// TIA Portal V15.1 export
// export: Created 2024-06-21T08:41:02.9041291Z, ExportSetting WithDefaults, DisplayName Totally Integrated Automation Portal, DisplayVersion V15.1 Update 5, DisplayName TIA Portal Openness, DisplayVersion V15.1 Update 5, DisplayName SINAMICS Startdrive Advanced, DisplayVersion V15.1, DisplayName G130, G150, S120, S150, SINAMICS MV, S210, DisplayVersion V15.1, DisplayName G110M, G120, G120C, G120D, G120P, DisplayVersion V15.1, DisplayName STEP 7 Professional, DisplayVersion V15.1 Update 5, DisplayName STEP 7 Safety, DisplayVersion V15.1, DisplayName WinCC Professional, DisplayVersion V15.1 Update 5, DisplayName SIMATIC Visualization Architect, DisplayVersion V15.1
FUNCTION_BLOCK "LProcModesSum"   // FB1702, FBD
TITLE = LProcModesSum
{ S7_Optimized_Access := 'FALSE' }
AUTHOR : VCC
FAMILY : ProcEqp
NAME : ModesSum
VERSION : 1.0
// ================================================================================
// Create the Modes Summary for 20 possible components
// ================================================================================
// stored: AutoNumber false, IsIECCheckEnabled false, SetENOAutomatically False, UDAEnableTagReadback false
   VAR_INPUT
      I_StartPB { ExternalAccessible := 'False'; ExternalVisible := 'False'; ExternalWritable := 'False'} : Bool;   // Summary of Start buttons
      I_AlarmResetPB { ExternalAccessible := 'False'; ExternalVisible := 'False'; ExternalWritable := 'False'} : Bool;   // Summary of Alarm reset buttons
      I_SafetyNotOk { ExternalAccessible := 'False'; ExternalVisible := 'False'; ExternalWritable := 'False'} : Bool;   // Safety is not ok
      I_ObjectMode1 { ExternalAccessible := 'False'; ExternalVisible := 'False'; ExternalWritable := 'False'} : Word;   // Modes Component 1
      I_ObjectMode2 { ExternalAccessible := 'False'; ExternalVisible := 'False'; ExternalWritable := 'False'} : Word;   // Modes Component 2
      I_ObjectMode3 { ExternalAccessible := 'False'; ExternalVisible := 'False'; ExternalWritable := 'False'} : Word;   // Modes Component 3
      I_ObjectMode3Used { ExternalAccessible := 'False'; ExternalVisible := 'False'; ExternalWritable := 'False'} : Bool;   // True if used
      I_ObjectMode4 { ExternalAccessible := 'False'; ExternalVisible := 'False'; ExternalWritable := 'False'} : Word;   // Modes Component 4
      I_ObjectMode4Used { ExternalAccessible := 'False'; ExternalVisible := 'False'; ExternalWritable := 'False'} : Bool;   // True if used
      I_ObjectMode5 { ExternalAccessible := 'False'; ExternalVisible := 'False'; ExternalWritable := 'False'} : Word;   // Modes Component 5
      I_ObjectMode5Used { ExternalAccessible := 'False'; ExternalVisible := 'False'; ExternalWritable := 'False'} : Bool;   // True if used
      I_ObjectMode6 { ExternalAccessible := 'False'; ExternalVisible := 'False'; ExternalWritable := 'False'} : Word;   // Modes Component 6
      I_ObjectMode6Used { ExternalAccessible := 'False'; ExternalVisible := 'False'; ExternalWritable := 'False'} : Bool;   // True if used
      I_ObjectMode7 { ExternalAccessible := 'False'; ExternalVisible := 'False'; ExternalWritable := 'False'} : Word;   // Modes Component 7
      I_ObjectMode7Used { ExternalAccessible := 'False'; ExternalVisible := 'False'; ExternalWritable := 'False'} : Bool;   // True if used
      I_ObjectMode8 { ExternalAccessible := 'False'; ExternalVisible := 'False'; ExternalWritable := 'False'} : Word;   // Modes Component 8
      I_ObjectMode8Used { ExternalAccessible := 'False'; ExternalVisible := 'False'; ExternalWritable := 'False'} : Bool;   // True if used
      I_ObjectMode9 { ExternalAccessible := 'False'; ExternalVisible := 'False'; ExternalWritable := 'False'} : Word;   // Modes Component 9
      I_ObjectMode9Used { ExternalAccessible := 'False'; ExternalVisible := 'False'; ExternalWritable := 'False'} : Bool;   // True if used
      I_ObjectMode10 { ExternalAccessible := 'False'; ExternalVisible := 'False'; ExternalWritable := 'False'} : Word;   // Modes Component 10
      I_ObjectMode10Used { ExternalAccessible := 'False'; ExternalVisible := 'False'; ExternalWritable := 'False'} : Bool;   // True if used
      I_ObjectMode11 { ExternalAccessible := 'False'; ExternalVisible := 'False'; ExternalWritable := 'False'} : Word;   // Modes Component 11
      I_ObjectMode11Used { ExternalAccessible := 'False'; ExternalVisible := 'False'; ExternalWritable := 'False'} : Bool;   // True if used
      I_ObjectMode12 { ExternalAccessible := 'False'; ExternalVisible := 'False'; ExternalWritable := 'False'} : Word;   // Modes Component 12
      I_ObjectMode12Used { ExternalAccessible := 'False'; ExternalVisible := 'False'; ExternalWritable := 'False'} : Bool;   // True if used
      I_ObjectMode13 { ExternalAccessible := 'False'; ExternalVisible := 'False'; ExternalWritable := 'False'} : Word;   // Modes Component 13
      I_ObjectMode13Used { ExternalAccessible := 'False'; ExternalVisible := 'False'; ExternalWritable := 'False'} : Bool;   // True if used
      I_ObjectMode14 { ExternalAccessible := 'False'; ExternalVisible := 'False'; ExternalWritable := 'False'} : Word;   // Modes Component 14
      I_ObjectMode14Used { ExternalAccessible := 'False'; ExternalVisible := 'False'; ExternalWritable := 'False'} : Bool;   // True if used
      I_ObjectMode15 { ExternalAccessible := 'False'; ExternalVisible := 'False'; ExternalWritable := 'False'} : Word;   // Modes Component 15
      I_ObjectMode15Used { ExternalAccessible := 'False'; ExternalVisible := 'False'; ExternalWritable := 'False'} : Bool;   // True if used
      I_ObjectMode16 { ExternalAccessible := 'False'; ExternalVisible := 'False'; ExternalWritable := 'False'} : Word;   // Modes Component 16
      I_ObjectMode16Used { ExternalAccessible := 'False'; ExternalVisible := 'False'; ExternalWritable := 'False'} : Bool;   // True if used
      I_ObjectMode17 { ExternalAccessible := 'False'; ExternalVisible := 'False'; ExternalWritable := 'False'} : Word;   // Modes Component 17
      I_ObjectMode17Used { ExternalAccessible := 'False'; ExternalVisible := 'False'; ExternalWritable := 'False'} : Bool;   // True if used
      I_ObjectMode18 { ExternalAccessible := 'False'; ExternalVisible := 'False'; ExternalWritable := 'False'} : Word;   // Modes Component 18
      I_ObjectMode18Used { ExternalAccessible := 'False'; ExternalVisible := 'False'; ExternalWritable := 'False'} : Bool;   // True if used
      I_ObjectMode19 { ExternalAccessible := 'False'; ExternalVisible := 'False'; ExternalWritable := 'False'} : Word;   // Modes Component 19
      I_ObjectMode19Used { ExternalAccessible := 'False'; ExternalVisible := 'False'; ExternalWritable := 'False'} : Bool;   // True if used
      I_ObjectMode20 { ExternalAccessible := 'False'; ExternalVisible := 'False'; ExternalWritable := 'False'} : Word;   // Modes Component 20
      I_ObjectMode20Used { ExternalAccessible := 'False'; ExternalVisible := 'False'; ExternalWritable := 'False'} : Bool;   // True if used
   END_VAR
   VAR_OUTPUT
      O_AutoSel { ExternalAccessible := 'False'; ExternalVisible := 'False'; ExternalWritable := 'False'} : Bool;   // At least one component is in auto selected
      O_Auto { ExternalAccessible := 'False'; ExternalVisible := 'False'; ExternalWritable := 'False'} : Bool;   // All the components are in auto
      O_ManSel { ExternalAccessible := 'False'; ExternalVisible := 'False'; ExternalWritable := 'False'} : Bool;   // At least one component is in manual selected
      O_Man { ExternalAccessible := 'False'; ExternalVisible := 'False'; ExternalWritable := 'False'} : Bool;   // At least one component is in manual
      O_AlarmResetPB { ExternalAccessible := 'False'; ExternalVisible := 'False'; ExternalWritable := 'False'} : Bool;   // Alarm reset button is activated
   END_VAR
   VAR DB_SPECIFIC
      H_Anim : Word;   // Mode Animation Word
      H_Anim2 : Word;   // Mode Animation Word
      H_ConfigBtnResetTM : Bool;   // From the HMI - Config internal tag
      H_ConfigBtnResetSeq : Bool;   // From the HMI - Config internal tag
      H_ModeChanged : Bool;   // From the HMI - Mode changed to Auto
      H_ScreenChanged : Bool;   // From the HMI - The screen has changed
      AutoSel1 { ExternalAccessible := 'False'; ExternalVisible := 'False'; ExternalWritable := 'False'} : Bool;   // Auto selected Component 1
      Auto1 { ExternalAccessible := 'False'; ExternalVisible := 'False'; ExternalWritable := 'False'} : Bool;   // Auto Component 1
      ManSel1 { ExternalAccessible := 'False'; ExternalVisible := 'False'; ExternalWritable := 'False'} : Bool;   // Manu selected Component 1
      Man1 { ExternalAccessible := 'False'; ExternalVisible := 'False'; ExternalWritable := 'False'} : Bool;   // Manu Component 1
      AutoSel2 { ExternalAccessible := 'False'; ExternalVisible := 'False'; ExternalWritable := 'False'} : Bool;   // Auto selected Component 2
      Auto2 { ExternalAccessible := 'False'; ExternalVisible := 'False'; ExternalWritable := 'False'} : Bool;   // Auto Component 2
      ManSel2 { ExternalAccessible := 'False'; ExternalVisible := 'False'; ExternalWritable := 'False'} : Bool;   // Manu selected Component 2
      Man2 { ExternalAccessible := 'False'; ExternalVisible := 'False'; ExternalWritable := 'False'} : Bool;   // Manu Component 2
      AutoSel3 { ExternalAccessible := 'False'; ExternalVisible := 'False'; ExternalWritable := 'False'} : Bool;   // Auto selected Component 3
      Auto3 { ExternalAccessible := 'False'; ExternalVisible := 'False'; ExternalWritable := 'False'} : Bool;   // Auto Component 3
      ManSel3 { ExternalAccessible := 'False'; ExternalVisible := 'False'; ExternalWritable := 'False'} : Bool;   // Manu selected Component 3
      Man3 { ExternalAccessible := 'False'; ExternalVisible := 'False'; ExternalWritable := 'False'} : Bool;   // Manu Component 3
      AutoSel4 { ExternalAccessible := 'False'; ExternalVisible := 'False'; ExternalWritable := 'False'} : Bool;   // Auto selected Component 4
      Auto4 { ExternalAccessible := 'False'; ExternalVisible := 'False'; ExternalWritable := 'False'} : Bool;   // Auto Component 4
      ManSel4 { ExternalAccessible := 'False'; ExternalVisible := 'False'; ExternalWritable := 'False'} : Bool;   // Manu selected Component 4
      Man4 { ExternalAccessible := 'False'; ExternalVisible := 'False'; ExternalWritable := 'False'} : Bool;   // Manu Component 4
      AutoSel5 { ExternalAccessible := 'False'; ExternalVisible := 'False'; ExternalWritable := 'False'} : Bool;   // Auto selected Component 5
      Auto5 { ExternalAccessible := 'False'; ExternalVisible := 'False'; ExternalWritable := 'False'} : Bool;   // Auto Component 5
      ManSel5 { ExternalAccessible := 'False'; ExternalVisible := 'False'; ExternalWritable := 'False'} : Bool;   // Manu selected Component 5
      Man5 { ExternalAccessible := 'False'; ExternalVisible := 'False'; ExternalWritable := 'False'} : Bool;   // Manu Component 5
      AutoSel6 { ExternalAccessible := 'False'; ExternalVisible := 'False'; ExternalWritable := 'False'} : Bool;   // Auto selected Component 6
      Auto6 { ExternalAccessible := 'False'; ExternalVisible := 'False'; ExternalWritable := 'False'} : Bool;   // Auto Component 6
      ManSel6 { ExternalAccessible := 'False'; ExternalVisible := 'False'; ExternalWritable := 'False'} : Bool;   // Manu selected Component 6
      Man6 { ExternalAccessible := 'False'; ExternalVisible := 'False'; ExternalWritable := 'False'} : Bool;   // Manu Component 6
      AutoSel7 { ExternalAccessible := 'False'; ExternalVisible := 'False'; ExternalWritable := 'False'} : Bool;   // Auto selected Component 7
      Auto7 { ExternalAccessible := 'False'; ExternalVisible := 'False'; ExternalWritable := 'False'} : Bool;   // Auto Component 7
      ManSel7 { ExternalAccessible := 'False'; ExternalVisible := 'False'; ExternalWritable := 'False'} : Bool;   // Manu selected Component 7
      Man7 { ExternalAccessible := 'False'; ExternalVisible := 'False'; ExternalWritable := 'False'} : Bool;   // Manu Component 7
      AutoSel8 { ExternalAccessible := 'False'; ExternalVisible := 'False'; ExternalWritable := 'False'} : Bool;   // Auto selected Component 8
      Auto8 { ExternalAccessible := 'False'; ExternalVisible := 'False'; ExternalWritable := 'False'} : Bool;   // Auto Component 8
      ManSel8 { ExternalAccessible := 'False'; ExternalVisible := 'False'; ExternalWritable := 'False'} : Bool;   // Manu selected Component 8
      Man8 { ExternalAccessible := 'False'; ExternalVisible := 'False'; ExternalWritable := 'False'} : Bool;   // Manu Component 8
      AutoSel9 { ExternalAccessible := 'False'; ExternalVisible := 'False'; ExternalWritable := 'False'} : Bool;   // Auto selected Component 9
      Auto9 { ExternalAccessible := 'False'; ExternalVisible := 'False'; ExternalWritable := 'False'} : Bool;   // Auto Component 9
      ManSel9 { ExternalAccessible := 'False'; ExternalVisible := 'False'; ExternalWritable := 'False'} : Bool;   // Manu selected Component 9
      Man9 { ExternalAccessible := 'False'; ExternalVisible := 'False'; ExternalWritable := 'False'} : Bool;   // Manu Component 9
      AutoSel10 { ExternalAccessible := 'False'; ExternalVisible := 'False'; ExternalWritable := 'False'} : Bool;   // Auto selected Component 10
      Auto10 { ExternalAccessible := 'False'; ExternalVisible := 'False'; ExternalWritable := 'False'} : Bool;   // Auto Component 10
      ManSel10 { ExternalAccessible := 'False'; ExternalVisible := 'False'; ExternalWritable := 'False'} : Bool;   // Manu selected Component 10
      Man10 { ExternalAccessible := 'False'; ExternalVisible := 'False'; ExternalWritable := 'False'} : Bool;   // Manu Component 10
      AutoSel11 { ExternalAccessible := 'False'; ExternalVisible := 'False'; ExternalWritable := 'False'} : Bool;   // Auto selected Component 11
      Auto11 { ExternalAccessible := 'False'; ExternalVisible := 'False'; ExternalWritable := 'False'} : Bool;   // Auto Component 11
      ManSel11 { ExternalAccessible := 'False'; ExternalVisible := 'False'; ExternalWritable := 'False'} : Bool;   // Manu selected Component 11
      Man11 { ExternalAccessible := 'False'; ExternalVisible := 'False'; ExternalWritable := 'False'} : Bool;   // Manu Component 11
      AutoSel12 { ExternalAccessible := 'False'; ExternalVisible := 'False'; ExternalWritable := 'False'} : Bool;   // Auto selected Component 12
      Auto12 { ExternalAccessible := 'False'; ExternalVisible := 'False'; ExternalWritable := 'False'} : Bool;   // Auto Component 12
      ManSel12 { ExternalAccessible := 'False'; ExternalVisible := 'False'; ExternalWritable := 'False'} : Bool;   // Manu selected Component 12
      Man12 { ExternalAccessible := 'False'; ExternalVisible := 'False'; ExternalWritable := 'False'} : Bool;   // Manu Component 12
      AutoSel13 { ExternalAccessible := 'False'; ExternalVisible := 'False'; ExternalWritable := 'False'} : Bool;   // Auto selected Component 13
      Auto13 { ExternalAccessible := 'False'; ExternalVisible := 'False'; ExternalWritable := 'False'} : Bool;   // Auto Component 13
      ManSel13 { ExternalAccessible := 'False'; ExternalVisible := 'False'; ExternalWritable := 'False'} : Bool;   // Manu selected Component 13
      Man13 { ExternalAccessible := 'False'; ExternalVisible := 'False'; ExternalWritable := 'False'} : Bool;   // Manu Component 13
      AutoSel14 { ExternalAccessible := 'False'; ExternalVisible := 'False'; ExternalWritable := 'False'} : Bool;   // Auto selected Component 14
      Auto14 { ExternalAccessible := 'False'; ExternalVisible := 'False'; ExternalWritable := 'False'} : Bool;   // Auto Component 14
      ManSel14 { ExternalAccessible := 'False'; ExternalVisible := 'False'; ExternalWritable := 'False'} : Bool;   // Manu selected Component 14
      Man14 { ExternalAccessible := 'False'; ExternalVisible := 'False'; ExternalWritable := 'False'} : Bool;   // Manu Component 14
      AutoSel15 { ExternalAccessible := 'False'; ExternalVisible := 'False'; ExternalWritable := 'False'} : Bool;   // Auto selected Component 15
      Auto15 { ExternalAccessible := 'False'; ExternalVisible := 'False'; ExternalWritable := 'False'} : Bool;   // Auto Component 15
      ManSel15 { ExternalAccessible := 'False'; ExternalVisible := 'False'; ExternalWritable := 'False'} : Bool;   // Manu selected Component 15
      Man15 { ExternalAccessible := 'False'; ExternalVisible := 'False'; ExternalWritable := 'False'} : Bool;   // Manu Component 15
      AutoSel16 { ExternalAccessible := 'False'; ExternalVisible := 'False'; ExternalWritable := 'False'} : Bool;   // Auto selected Component 16
      Auto16 { ExternalAccessible := 'False'; ExternalVisible := 'False'; ExternalWritable := 'False'} : Bool;   // Auto Component 16
      ManSel16 { ExternalAccessible := 'False'; ExternalVisible := 'False'; ExternalWritable := 'False'} : Bool;   // Manu selected Component 16
      Man16 { ExternalAccessible := 'False'; ExternalVisible := 'False'; ExternalWritable := 'False'} : Bool;   // Manu Component 16
      AutoSel17 { ExternalAccessible := 'False'; ExternalVisible := 'False'; ExternalWritable := 'False'} : Bool;   // Auto selected Component 17
      Auto17 { ExternalAccessible := 'False'; ExternalVisible := 'False'; ExternalWritable := 'False'} : Bool;   // Auto Component 17
      ManSel17 { ExternalAccessible := 'False'; ExternalVisible := 'False'; ExternalWritable := 'False'} : Bool;   // Manu selected Component 17
      Man17 { ExternalAccessible := 'False'; ExternalVisible := 'False'; ExternalWritable := 'False'} : Bool;   // Manu Component 17
      AutoSel18 { ExternalAccessible := 'False'; ExternalVisible := 'False'; ExternalWritable := 'False'} : Bool;   // Auto selected Component 18
      Auto18 { ExternalAccessible := 'False'; ExternalVisible := 'False'; ExternalWritable := 'False'} : Bool;   // Auto Component 18
      ManSel18 { ExternalAccessible := 'False'; ExternalVisible := 'False'; ExternalWritable := 'False'} : Bool;   // Manu selected Component 18
      Man18 { ExternalAccessible := 'False'; ExternalVisible := 'False'; ExternalWritable := 'False'} : Bool;   // Manu Component 18
      AutoSel19 { ExternalAccessible := 'False'; ExternalVisible := 'False'; ExternalWritable := 'False'} : Bool;   // Auto selected Component 19
      Auto19 { ExternalAccessible := 'False'; ExternalVisible := 'False'; ExternalWritable := 'False'} : Bool;   // Auto Component 19
      ManSel19 { ExternalAccessible := 'False'; ExternalVisible := 'False'; ExternalWritable := 'False'} : Bool;   // Manu selected Component 19
      Man19 { ExternalAccessible := 'False'; ExternalVisible := 'False'; ExternalWritable := 'False'} : Bool;   // Manu Component 19
      AutoSel20 { ExternalAccessible := 'False'; ExternalVisible := 'False'; ExternalWritable := 'False'} : Bool;   // Auto selected Component 20
      Auto20 { ExternalAccessible := 'False'; ExternalVisible := 'False'; ExternalWritable := 'False'} : Bool;   // Auto Component 20
      ManSel20 { ExternalAccessible := 'False'; ExternalVisible := 'False'; ExternalWritable := 'False'} : Bool;   // Manu selected Component 20
      Man20 { ExternalAccessible := 'False'; ExternalVisible := 'False'; ExternalWritable := 'False'} : Bool;   // Manu Component 20
      Auto { ExternalAccessible := 'False'; ExternalVisible := 'False'; ExternalWritable := 'False'} : Bool;   // Auto Mode Summary
      Man { ExternalAccessible := 'False'; ExternalVisible := 'False'; ExternalWritable := 'False'} : Bool;   // Manual Mode Summary
      AutoSel { ExternalAccessible := 'False'; ExternalVisible := 'False'; ExternalWritable := 'False'} : Bool;   // Auto Mode Selected Summary
      ManSel { ExternalAccessible := 'False'; ExternalVisible := 'False'; ExternalWritable := 'False'} : Bool;   // Manual Mode Selected Summary
      TimerStartPBSel { ExternalAccessible := 'False'; ExternalVisible := 'False'; ExternalWritable := 'False'; S7_SetPoint := 'True'} : TOF_TIME;   // Timer
      TimerAlarmResetPBSel { ExternalAccessible := 'False'; ExternalVisible := 'False'; ExternalWritable := 'False'; S7_SetPoint := 'True'} : TOF_TIME;   // Timer
   END_VAR
BEGIN

REGION Network 1: **** 1 - Inputs **** Extract Mode Component 1
   // Extract Mode Component 1
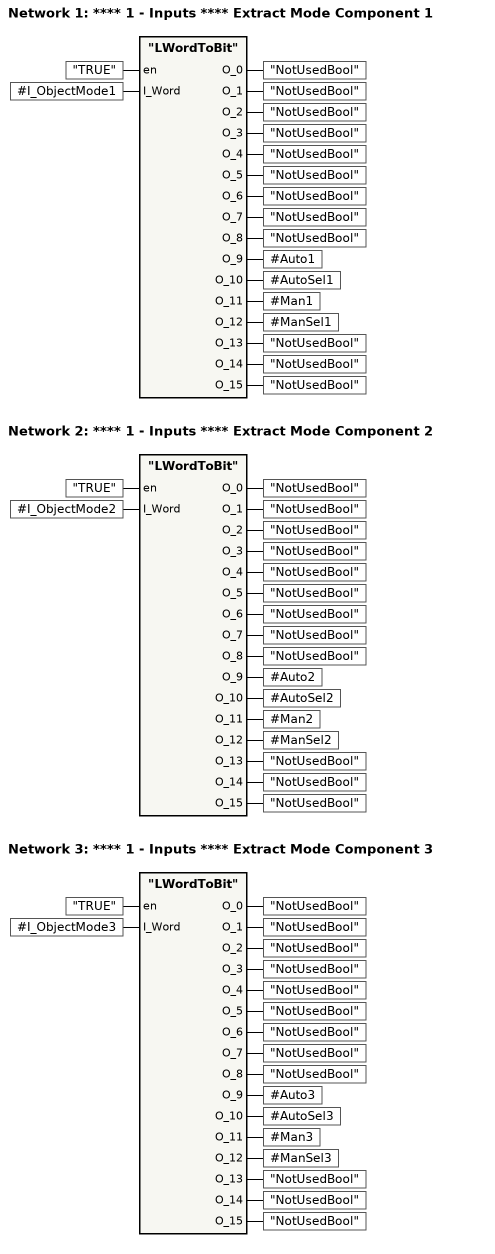
   IF "TRUE" THEN
       "LWordToBit"(I_Word := #I_ObjectMode1,
                    O_0 => "NotUsedBool",
                    O_1 => "NotUsedBool",
                    O_2 => "NotUsedBool",
                    O_3 => "NotUsedBool",
                    O_4 => "NotUsedBool",
                    O_5 => "NotUsedBool",
                    O_6 => "NotUsedBool",
                    O_7 => "NotUsedBool",
                    O_8 => "NotUsedBool",
                    O_9 => #Auto1,
                    O_10 => #AutoSel1,
                    O_11 => #Man1,
                    O_12 => #ManSel1,
                    O_13 => "NotUsedBool",
                    O_14 => "NotUsedBool",
                    O_15 => "NotUsedBool");
   END_IF;
END_REGION

REGION Network 2: **** 1 - Inputs **** Extract Mode Component 2
   // Extract Mode Component 2
   IF "TRUE" THEN
       "LWordToBit"(I_Word := #I_ObjectMode2,
                    O_0 => "NotUsedBool",
                    O_1 => "NotUsedBool",
                    O_2 => "NotUsedBool",
                    O_3 => "NotUsedBool",
                    O_4 => "NotUsedBool",
                    O_5 => "NotUsedBool",
                    O_6 => "NotUsedBool",
                    O_7 => "NotUsedBool",
                    O_8 => "NotUsedBool",
                    O_9 => #Auto2,
                    O_10 => #AutoSel2,
                    O_11 => #Man2,
                    O_12 => #ManSel2,
                    O_13 => "NotUsedBool",
                    O_14 => "NotUsedBool",
                    O_15 => "NotUsedBool");
   END_IF;
END_REGION

REGION Network 3: **** 1 - Inputs **** Extract Mode Component 3
   // Extract Mode Component 3
   IF "TRUE" THEN
       "LWordToBit"(I_Word := #I_ObjectMode3,
                    O_0 => "NotUsedBool",
                    O_1 => "NotUsedBool",
                    O_2 => "NotUsedBool",
                    O_3 => "NotUsedBool",
                    O_4 => "NotUsedBool",
                    O_5 => "NotUsedBool",
                    O_6 => "NotUsedBool",
                    O_7 => "NotUsedBool",
                    O_8 => "NotUsedBool",
                    O_9 => #Auto3,
                    O_10 => #AutoSel3,
                    O_11 => #Man3,
                    O_12 => #ManSel3,
                    O_13 => "NotUsedBool",
                    O_14 => "NotUsedBool",
                    O_15 => "NotUsedBool");
   END_IF;
END_REGION

REGION Network 4: **** 1 - Inputs **** Extract Mode Component 4
   // Extract Mode Component 4
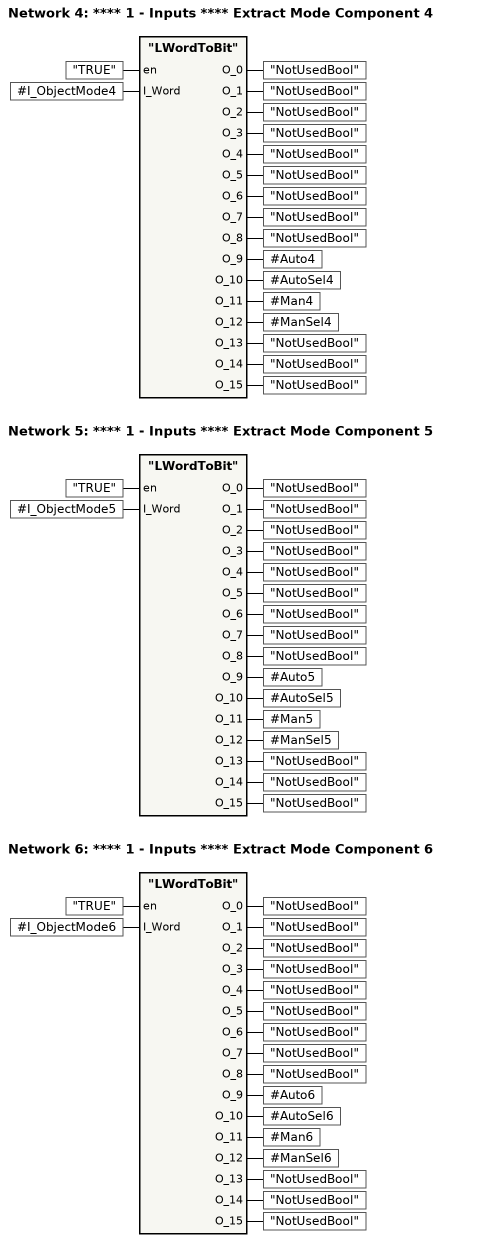
   IF "TRUE" THEN
       "LWordToBit"(I_Word := #I_ObjectMode4,
                    O_0 => "NotUsedBool",
                    O_1 => "NotUsedBool",
                    O_2 => "NotUsedBool",
                    O_3 => "NotUsedBool",
                    O_4 => "NotUsedBool",
                    O_5 => "NotUsedBool",
                    O_6 => "NotUsedBool",
                    O_7 => "NotUsedBool",
                    O_8 => "NotUsedBool",
                    O_9 => #Auto4,
                    O_10 => #AutoSel4,
                    O_11 => #Man4,
                    O_12 => #ManSel4,
                    O_13 => "NotUsedBool",
                    O_14 => "NotUsedBool",
                    O_15 => "NotUsedBool");
   END_IF;
END_REGION

REGION Network 5: **** 1 - Inputs **** Extract Mode Component 5
   // Extract Mode Component 5
   IF "TRUE" THEN
       "LWordToBit"(I_Word := #I_ObjectMode5,
                    O_0 => "NotUsedBool",
                    O_1 => "NotUsedBool",
                    O_2 => "NotUsedBool",
                    O_3 => "NotUsedBool",
                    O_4 => "NotUsedBool",
                    O_5 => "NotUsedBool",
                    O_6 => "NotUsedBool",
                    O_7 => "NotUsedBool",
                    O_8 => "NotUsedBool",
                    O_9 => #Auto5,
                    O_10 => #AutoSel5,
                    O_11 => #Man5,
                    O_12 => #ManSel5,
                    O_13 => "NotUsedBool",
                    O_14 => "NotUsedBool",
                    O_15 => "NotUsedBool");
   END_IF;
END_REGION

REGION Network 6: **** 1 - Inputs **** Extract Mode Component 6
   // Extract Mode Component 6
   IF "TRUE" THEN
       "LWordToBit"(I_Word := #I_ObjectMode6,
                    O_0 => "NotUsedBool",
                    O_1 => "NotUsedBool",
                    O_2 => "NotUsedBool",
                    O_3 => "NotUsedBool",
                    O_4 => "NotUsedBool",
                    O_5 => "NotUsedBool",
                    O_6 => "NotUsedBool",
                    O_7 => "NotUsedBool",
                    O_8 => "NotUsedBool",
                    O_9 => #Auto6,
                    O_10 => #AutoSel6,
                    O_11 => #Man6,
                    O_12 => #ManSel6,
                    O_13 => "NotUsedBool",
                    O_14 => "NotUsedBool",
                    O_15 => "NotUsedBool");
   END_IF;
END_REGION

REGION Network 7: **** 1 - Inputs **** Extract Mode Component 7
   // Extract Mode Component 7
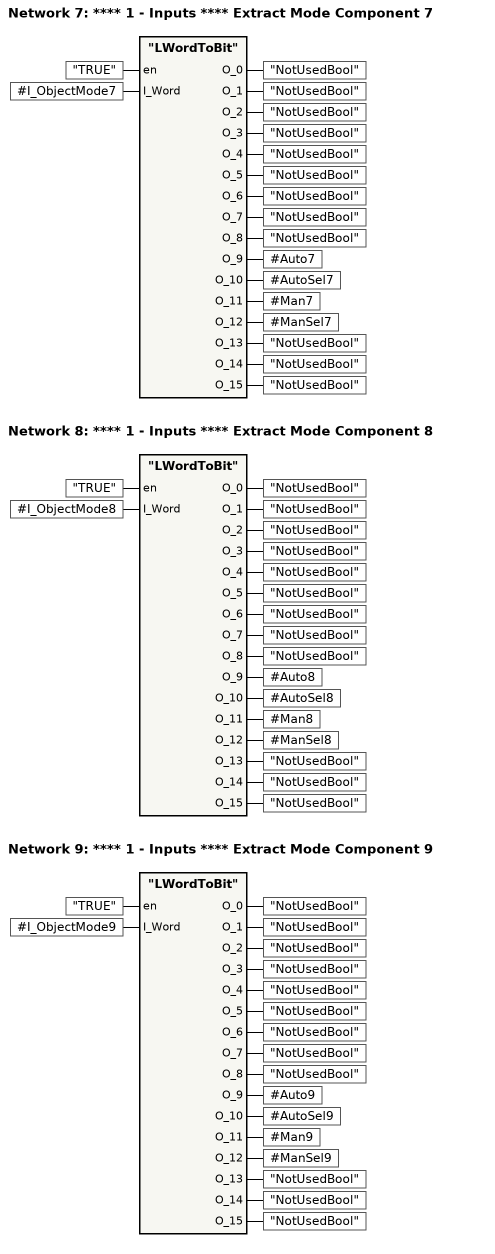
   IF "TRUE" THEN
       "LWordToBit"(I_Word := #I_ObjectMode7,
                    O_0 => "NotUsedBool",
                    O_1 => "NotUsedBool",
                    O_2 => "NotUsedBool",
                    O_3 => "NotUsedBool",
                    O_4 => "NotUsedBool",
                    O_5 => "NotUsedBool",
                    O_6 => "NotUsedBool",
                    O_7 => "NotUsedBool",
                    O_8 => "NotUsedBool",
                    O_9 => #Auto7,
                    O_10 => #AutoSel7,
                    O_11 => #Man7,
                    O_12 => #ManSel7,
                    O_13 => "NotUsedBool",
                    O_14 => "NotUsedBool",
                    O_15 => "NotUsedBool");
   END_IF;
END_REGION

REGION Network 8: **** 1 - Inputs **** Extract Mode Component 8
   // Extract Mode Component 8
   IF "TRUE" THEN
       "LWordToBit"(I_Word := #I_ObjectMode8,
                    O_0 => "NotUsedBool",
                    O_1 => "NotUsedBool",
                    O_2 => "NotUsedBool",
                    O_3 => "NotUsedBool",
                    O_4 => "NotUsedBool",
                    O_5 => "NotUsedBool",
                    O_6 => "NotUsedBool",
                    O_7 => "NotUsedBool",
                    O_8 => "NotUsedBool",
                    O_9 => #Auto8,
                    O_10 => #AutoSel8,
                    O_11 => #Man8,
                    O_12 => #ManSel8,
                    O_13 => "NotUsedBool",
                    O_14 => "NotUsedBool",
                    O_15 => "NotUsedBool");
   END_IF;
END_REGION

REGION Network 9: **** 1 - Inputs **** Extract Mode Component 9
   // Extract Mode Component 9
   IF "TRUE" THEN
       "LWordToBit"(I_Word := #I_ObjectMode9,
                    O_0 => "NotUsedBool",
                    O_1 => "NotUsedBool",
                    O_2 => "NotUsedBool",
                    O_3 => "NotUsedBool",
                    O_4 => "NotUsedBool",
                    O_5 => "NotUsedBool",
                    O_6 => "NotUsedBool",
                    O_7 => "NotUsedBool",
                    O_8 => "NotUsedBool",
                    O_9 => #Auto9,
                    O_10 => #AutoSel9,
                    O_11 => #Man9,
                    O_12 => #ManSel9,
                    O_13 => "NotUsedBool",
                    O_14 => "NotUsedBool",
                    O_15 => "NotUsedBool");
   END_IF;
END_REGION

REGION Network 10: **** 1 - Inputs **** Extract Mode Component 10
   // Extract Mode Component 10
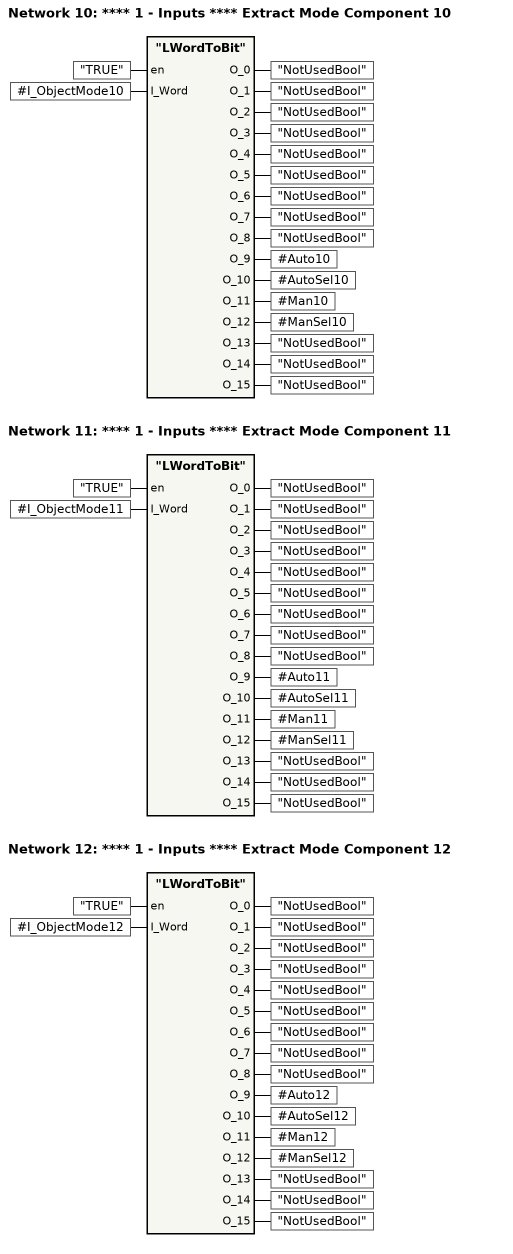
   IF "TRUE" THEN
       "LWordToBit"(I_Word := #I_ObjectMode10,
                    O_0 => "NotUsedBool",
                    O_1 => "NotUsedBool",
                    O_2 => "NotUsedBool",
                    O_3 => "NotUsedBool",
                    O_4 => "NotUsedBool",
                    O_5 => "NotUsedBool",
                    O_6 => "NotUsedBool",
                    O_7 => "NotUsedBool",
                    O_8 => "NotUsedBool",
                    O_9 => #Auto10,
                    O_10 => #AutoSel10,
                    O_11 => #Man10,
                    O_12 => #ManSel10,
                    O_13 => "NotUsedBool",
                    O_14 => "NotUsedBool",
                    O_15 => "NotUsedBool");
   END_IF;
END_REGION

REGION Network 11: **** 1 - Inputs **** Extract Mode Component 11
   // Extract Mode Component 11
   IF "TRUE" THEN
       "LWordToBit"(I_Word := #I_ObjectMode11,
                    O_0 => "NotUsedBool",
                    O_1 => "NotUsedBool",
                    O_2 => "NotUsedBool",
                    O_3 => "NotUsedBool",
                    O_4 => "NotUsedBool",
                    O_5 => "NotUsedBool",
                    O_6 => "NotUsedBool",
                    O_7 => "NotUsedBool",
                    O_8 => "NotUsedBool",
                    O_9 => #Auto11,
                    O_10 => #AutoSel11,
                    O_11 => #Man11,
                    O_12 => #ManSel11,
                    O_13 => "NotUsedBool",
                    O_14 => "NotUsedBool",
                    O_15 => "NotUsedBool");
   END_IF;
END_REGION

REGION Network 12: **** 1 - Inputs **** Extract Mode Component 12
   // Extract Mode Component 12
   IF "TRUE" THEN
       "LWordToBit"(I_Word := #I_ObjectMode12,
                    O_0 => "NotUsedBool",
                    O_1 => "NotUsedBool",
                    O_2 => "NotUsedBool",
                    O_3 => "NotUsedBool",
                    O_4 => "NotUsedBool",
                    O_5 => "NotUsedBool",
                    O_6 => "NotUsedBool",
                    O_7 => "NotUsedBool",
                    O_8 => "NotUsedBool",
                    O_9 => #Auto12,
                    O_10 => #AutoSel12,
                    O_11 => #Man12,
                    O_12 => #ManSel12,
                    O_13 => "NotUsedBool",
                    O_14 => "NotUsedBool",
                    O_15 => "NotUsedBool");
   END_IF;
END_REGION

REGION Network 13: **** 1 - Inputs **** Extract Mode Component 13
   // Extract Mode Component 13
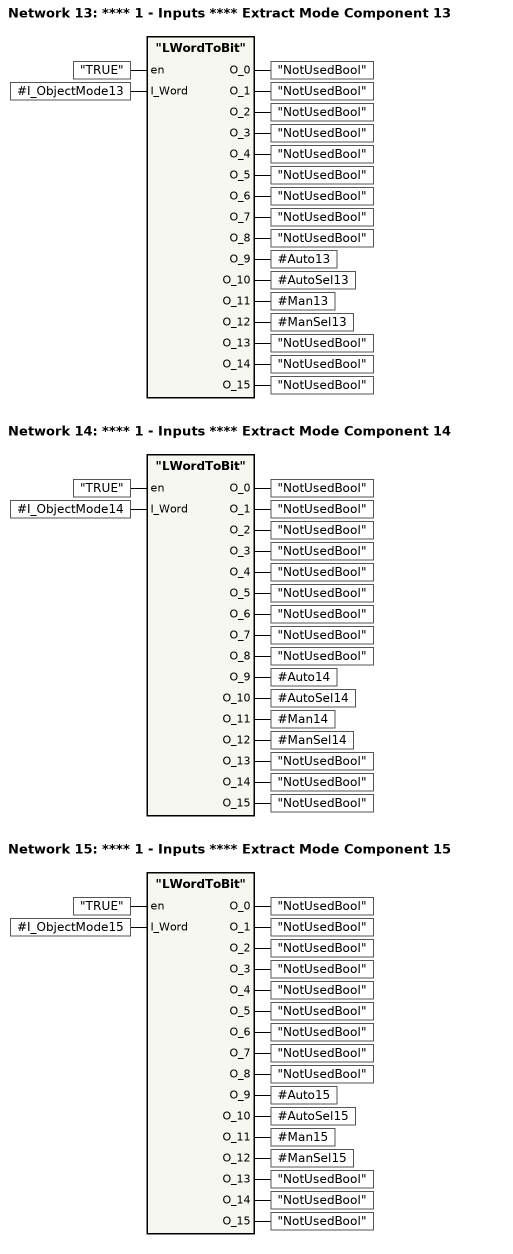
   IF "TRUE" THEN
       "LWordToBit"(I_Word := #I_ObjectMode13,
                    O_0 => "NotUsedBool",
                    O_1 => "NotUsedBool",
                    O_2 => "NotUsedBool",
                    O_3 => "NotUsedBool",
                    O_4 => "NotUsedBool",
                    O_5 => "NotUsedBool",
                    O_6 => "NotUsedBool",
                    O_7 => "NotUsedBool",
                    O_8 => "NotUsedBool",
                    O_9 => #Auto13,
                    O_10 => #AutoSel13,
                    O_11 => #Man13,
                    O_12 => #ManSel13,
                    O_13 => "NotUsedBool",
                    O_14 => "NotUsedBool",
                    O_15 => "NotUsedBool");
   END_IF;
END_REGION

REGION Network 14: **** 1 - Inputs **** Extract Mode Component 14
   // Extract Mode Component 14
   IF "TRUE" THEN
       "LWordToBit"(I_Word := #I_ObjectMode14,
                    O_0 => "NotUsedBool",
                    O_1 => "NotUsedBool",
                    O_2 => "NotUsedBool",
                    O_3 => "NotUsedBool",
                    O_4 => "NotUsedBool",
                    O_5 => "NotUsedBool",
                    O_6 => "NotUsedBool",
                    O_7 => "NotUsedBool",
                    O_8 => "NotUsedBool",
                    O_9 => #Auto14,
                    O_10 => #AutoSel14,
                    O_11 => #Man14,
                    O_12 => #ManSel14,
                    O_13 => "NotUsedBool",
                    O_14 => "NotUsedBool",
                    O_15 => "NotUsedBool");
   END_IF;
END_REGION

REGION Network 15: **** 1 - Inputs **** Extract Mode Component 15
   // Extract Mode Component 15
   IF "TRUE" THEN
       "LWordToBit"(I_Word := #I_ObjectMode15,
                    O_0 => "NotUsedBool",
                    O_1 => "NotUsedBool",
                    O_2 => "NotUsedBool",
                    O_3 => "NotUsedBool",
                    O_4 => "NotUsedBool",
                    O_5 => "NotUsedBool",
                    O_6 => "NotUsedBool",
                    O_7 => "NotUsedBool",
                    O_8 => "NotUsedBool",
                    O_9 => #Auto15,
                    O_10 => #AutoSel15,
                    O_11 => #Man15,
                    O_12 => #ManSel15,
                    O_13 => "NotUsedBool",
                    O_14 => "NotUsedBool",
                    O_15 => "NotUsedBool");
   END_IF;
END_REGION

REGION Network 16: **** 1 - Inputs **** Extract Mode Component 16
   // Extract Mode Component 16
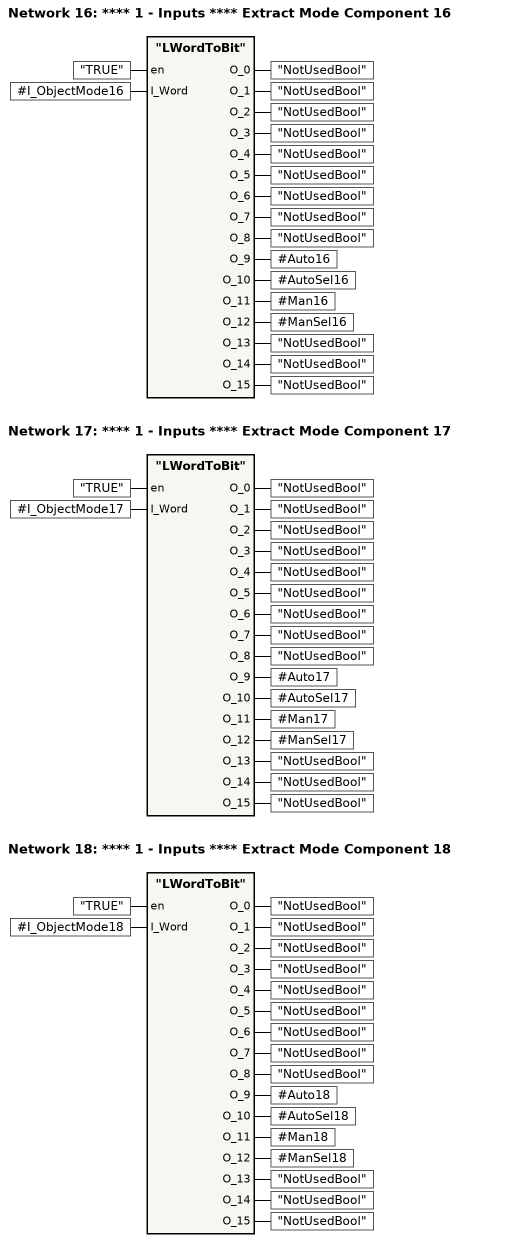
   IF "TRUE" THEN
       "LWordToBit"(I_Word := #I_ObjectMode16,
                    O_0 => "NotUsedBool",
                    O_1 => "NotUsedBool",
                    O_2 => "NotUsedBool",
                    O_3 => "NotUsedBool",
                    O_4 => "NotUsedBool",
                    O_5 => "NotUsedBool",
                    O_6 => "NotUsedBool",
                    O_7 => "NotUsedBool",
                    O_8 => "NotUsedBool",
                    O_9 => #Auto16,
                    O_10 => #AutoSel16,
                    O_11 => #Man16,
                    O_12 => #ManSel16,
                    O_13 => "NotUsedBool",
                    O_14 => "NotUsedBool",
                    O_15 => "NotUsedBool");
   END_IF;
END_REGION

REGION Network 17: **** 1 - Inputs **** Extract Mode Component 17
   // Extract Mode Component 17
   IF "TRUE" THEN
       "LWordToBit"(I_Word := #I_ObjectMode17,
                    O_0 => "NotUsedBool",
                    O_1 => "NotUsedBool",
                    O_2 => "NotUsedBool",
                    O_3 => "NotUsedBool",
                    O_4 => "NotUsedBool",
                    O_5 => "NotUsedBool",
                    O_6 => "NotUsedBool",
                    O_7 => "NotUsedBool",
                    O_8 => "NotUsedBool",
                    O_9 => #Auto17,
                    O_10 => #AutoSel17,
                    O_11 => #Man17,
                    O_12 => #ManSel17,
                    O_13 => "NotUsedBool",
                    O_14 => "NotUsedBool",
                    O_15 => "NotUsedBool");
   END_IF;
END_REGION

REGION Network 18: **** 1 - Inputs **** Extract Mode Component 18
   // Extract Mode Component 18
   IF "TRUE" THEN
       "LWordToBit"(I_Word := #I_ObjectMode18,
                    O_0 => "NotUsedBool",
                    O_1 => "NotUsedBool",
                    O_2 => "NotUsedBool",
                    O_3 => "NotUsedBool",
                    O_4 => "NotUsedBool",
                    O_5 => "NotUsedBool",
                    O_6 => "NotUsedBool",
                    O_7 => "NotUsedBool",
                    O_8 => "NotUsedBool",
                    O_9 => #Auto18,
                    O_10 => #AutoSel18,
                    O_11 => #Man18,
                    O_12 => #ManSel18,
                    O_13 => "NotUsedBool",
                    O_14 => "NotUsedBool",
                    O_15 => "NotUsedBool");
   END_IF;
END_REGION

REGION Network 19: **** 1 - Inputs **** Extract Mode Component 19
   // Extract Mode Component 19
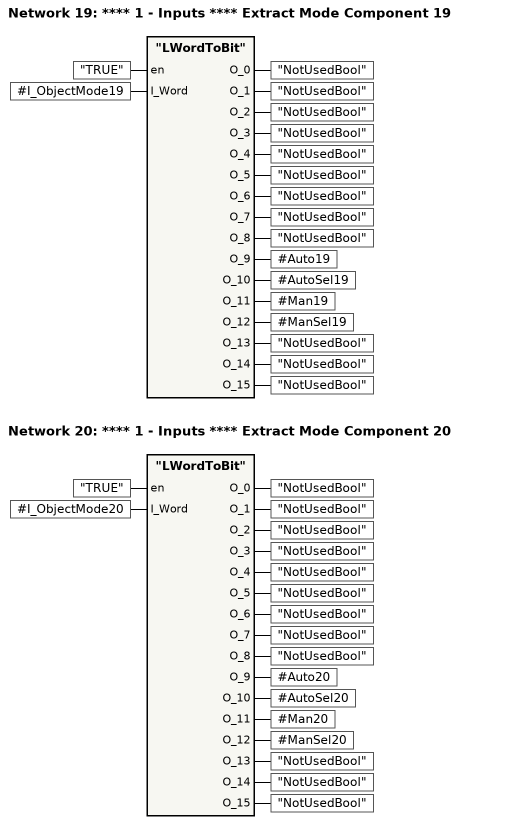
   IF "TRUE" THEN
       "LWordToBit"(I_Word := #I_ObjectMode19,
                    O_0 => "NotUsedBool",
                    O_1 => "NotUsedBool",
                    O_2 => "NotUsedBool",
                    O_3 => "NotUsedBool",
                    O_4 => "NotUsedBool",
                    O_5 => "NotUsedBool",
                    O_6 => "NotUsedBool",
                    O_7 => "NotUsedBool",
                    O_8 => "NotUsedBool",
                    O_9 => #Auto19,
                    O_10 => #AutoSel19,
                    O_11 => #Man19,
                    O_12 => #ManSel19,
                    O_13 => "NotUsedBool",
                    O_14 => "NotUsedBool",
                    O_15 => "NotUsedBool");
   END_IF;
END_REGION

REGION Network 20: **** 1 - Inputs **** Extract Mode Component 20
   // Extract Mode Component 20
   IF "TRUE" THEN
       "LWordToBit"(I_Word := #I_ObjectMode20,
                    O_0 => "NotUsedBool",
                    O_1 => "NotUsedBool",
                    O_2 => "NotUsedBool",
                    O_3 => "NotUsedBool",
                    O_4 => "NotUsedBool",
                    O_5 => "NotUsedBool",
                    O_6 => "NotUsedBool",
                    O_7 => "NotUsedBool",
                    O_8 => "NotUsedBool",
                    O_9 => #Auto20,
                    O_10 => #AutoSel20,
                    O_11 => #Man20,
                    O_12 => #ManSel20,
                    O_13 => "NotUsedBool",
                    O_14 => "NotUsedBool",
                    O_15 => "NotUsedBool");
   END_IF;
END_REGION

REGION Network 21: **** 4.6 - Machine status - Indications **** Summary Auto Mode
   // Summary Auto Mode
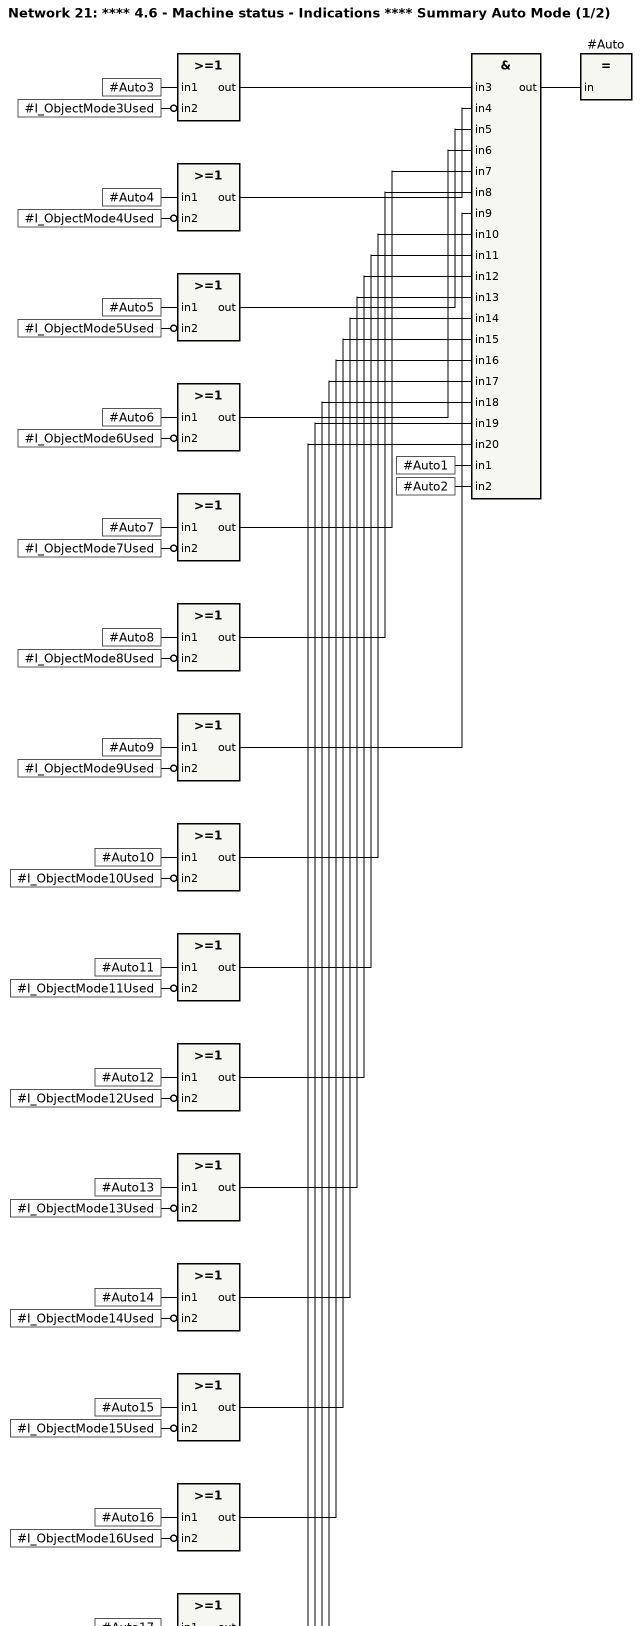
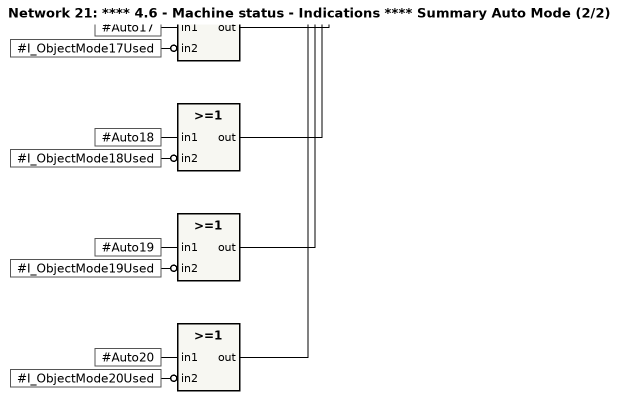
   #Auto := (#Auto3 OR NOT #I_ObjectMode3Used) AND (#Auto4 OR NOT #I_ObjectMode4Used) AND (#Auto5 OR NOT #I_ObjectMode5Used) AND (#Auto6 OR NOT #I_ObjectMode6Used) AND (#Auto7 OR NOT #I_ObjectMode7Used) AND (#Auto8 OR NOT #I_ObjectMode8Used) AND (#Auto9 OR NOT #I_ObjectMode9Used) AND (#Auto10 OR NOT #I_ObjectMode10Used) AND (#Auto11 OR NOT #I_ObjectMode11Used) AND (#Auto12 OR NOT #I_ObjectMode12Used) AND (#Auto13 OR NOT #I_ObjectMode13Used) AND (#Auto14 OR NOT #I_ObjectMode14Used) AND (#Auto15 OR NOT #I_ObjectMode15Used) AND (#Auto16 OR NOT #I_ObjectMode16Used) AND (#Auto17 OR NOT #I_ObjectMode17Used) AND (#Auto18 OR NOT #I_ObjectMode18Used) AND (#Auto19 OR NOT #I_ObjectMode19Used) AND (#Auto20 OR NOT #I_ObjectMode20Used) AND #Auto1 AND #Auto2;
END_REGION

REGION Network 22: **** 4.6 - Machine status - Indications **** Summary AutoSel
   // Summary AutoSel
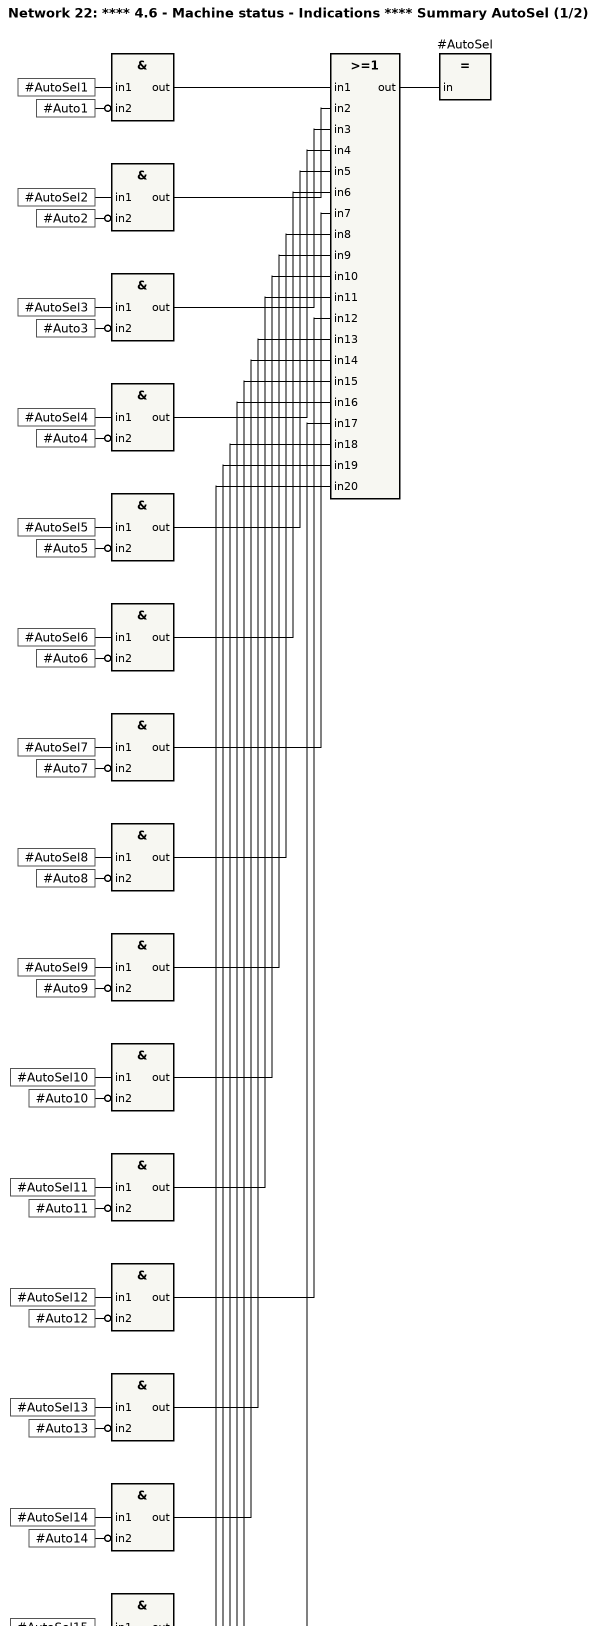
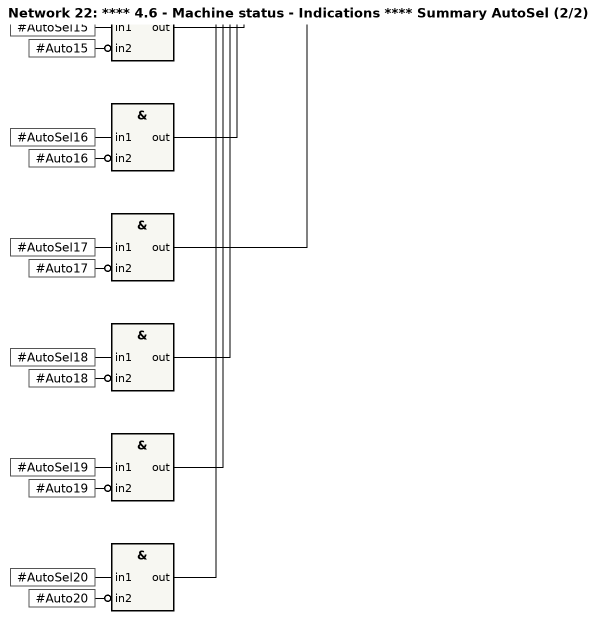
   #AutoSel := (#AutoSel1 AND NOT #Auto1) OR (#AutoSel2 AND NOT #Auto2) OR (#AutoSel3 AND NOT #Auto3) OR (#AutoSel4 AND NOT #Auto4) OR (#AutoSel5 AND NOT #Auto5) OR (#AutoSel6 AND NOT #Auto6) OR (#AutoSel7 AND NOT #Auto7) OR (#AutoSel8 AND NOT #Auto8) OR (#AutoSel9 AND NOT #Auto9) OR (#AutoSel10 AND NOT #Auto10) OR (#AutoSel11 AND NOT #Auto11) OR (#AutoSel12 AND NOT #Auto12) OR (#AutoSel13 AND NOT #Auto13) OR (#AutoSel14 AND NOT #Auto14) OR (#AutoSel15 AND NOT #Auto15) OR (#AutoSel16 AND NOT #Auto16) OR (#AutoSel17 AND NOT #Auto17) OR (#AutoSel18 AND NOT #Auto18) OR (#AutoSel19 AND NOT #Auto19) OR (#AutoSel20 AND NOT #Auto20);
END_REGION

REGION Network 23: **** 4.6 - Machine status - Indications **** Summary AutoSel
   // Summary AutoSel
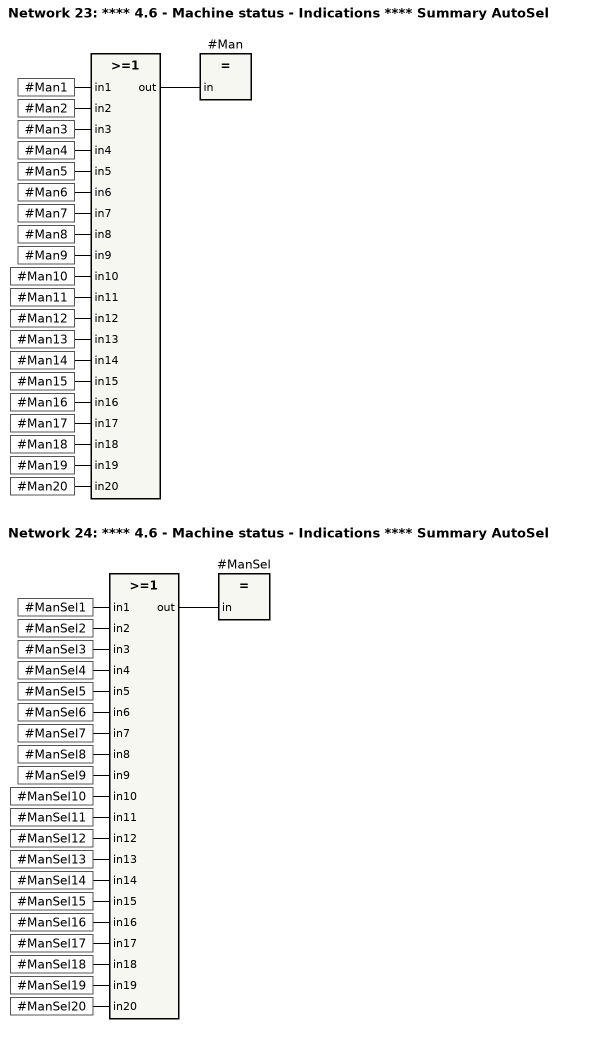
   #Man := #Man1 OR #Man2 OR #Man3 OR #Man4 OR #Man5 OR #Man6 OR #Man7 OR #Man8 OR #Man9 OR #Man10 OR #Man11 OR #Man12 OR #Man13 OR #Man14 OR #Man15 OR #Man16 OR #Man17 OR #Man18 OR #Man19 OR #Man20;
END_REGION

REGION Network 24: **** 4.6 - Machine status - Indications **** Summary AutoSel
   // Summary AutoSel
   #ManSel := #ManSel1 OR #ManSel2 OR #ManSel3 OR #ManSel4 OR #ManSel5 OR #ManSel6 OR #ManSel7 OR #ManSel8 OR #ManSel9 OR #ManSel10 OR #ManSel11 OR #ManSel12 OR #ManSel13 OR #ManSel14 OR #ManSel15 OR #ManSel16 OR #ManSel17 OR #ManSel18 OR #ManSel19 OR #ManSel20;
END_REGION

REGION Network 25: **** 4.6 - Machine Status - Indications **** Animation
   // Animation
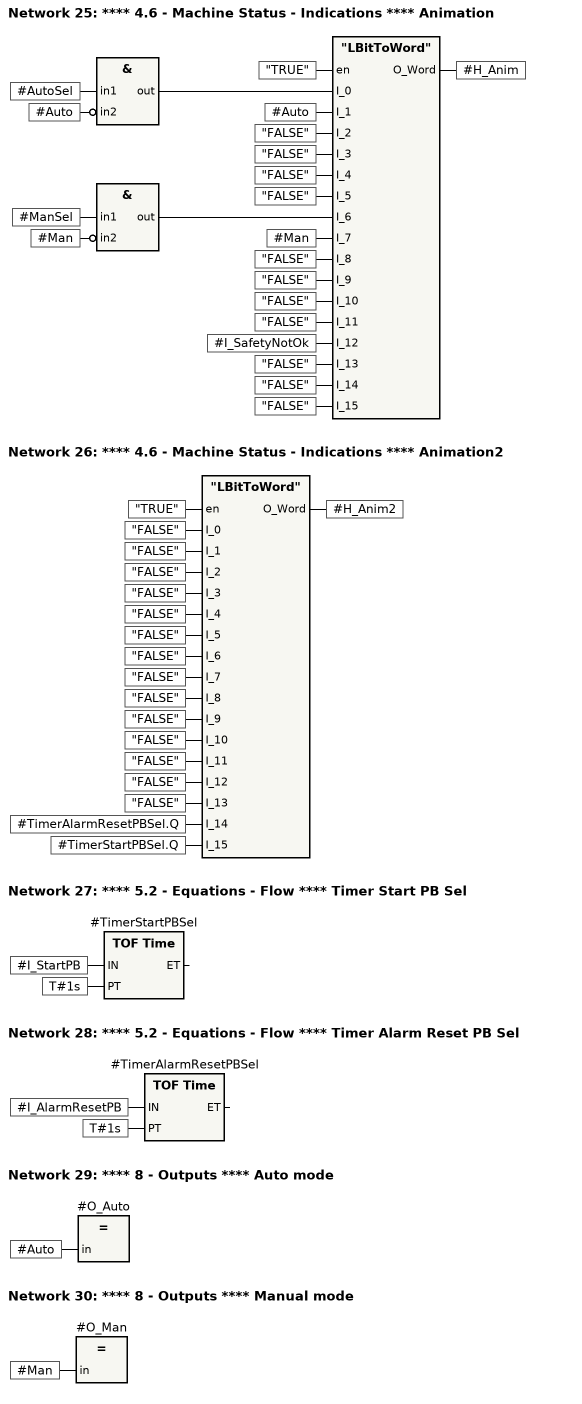
   IF "TRUE" THEN
       "LBitToWord"(I_0 := #AutoSel AND NOT #Auto,
                    I_1 := #Auto,
                    I_2 := "FALSE",
                    I_3 := "FALSE",
                    I_4 := "FALSE",
                    I_5 := "FALSE",
                    I_6 := #ManSel AND NOT #Man,
                    I_7 := #Man,
                    I_8 := "FALSE",
                    I_9 := "FALSE",
                    I_10 := "FALSE",
                    I_11 := "FALSE",
                    I_12 := #I_SafetyNotOk,
                    I_13 := "FALSE",
                    I_14 := "FALSE",
                    I_15 := "FALSE",
                    O_Word => #H_Anim);
   END_IF;
END_REGION

REGION Network 26: **** 4.6 - Machine Status - Indications **** Animation2
   // Animation
   IF "TRUE" THEN
       "LBitToWord"(I_0 := "FALSE",
                    I_1 := "FALSE",
                    I_2 := "FALSE",
                    I_3 := "FALSE",
                    I_4 := "FALSE",
                    I_5 := "FALSE",
                    I_6 := "FALSE",
                    I_7 := "FALSE",
                    I_8 := "FALSE",
                    I_9 := "FALSE",
                    I_10 := "FALSE",
                    I_11 := "FALSE",
                    I_12 := "FALSE",
                    I_13 := "FALSE",
                    I_14 := #TimerAlarmResetPBSel.Q,
                    I_15 := #TimerStartPBSel.Q,
                    O_Word => #H_Anim2);
   END_IF;
END_REGION

REGION Network 27: **** 5.2 - Equations - Flow **** Timer Start PB Sel
   // Timer Start PB Sel
   #TimerStartPBSel(IN := #I_StartPB, PT := T#1s);   // TOF
END_REGION

REGION Network 28: **** 5.2 - Equations - Flow **** Timer Alarm Reset PB Sel
   // Timer Alarm Reset PB Sel
   #TimerAlarmResetPBSel(IN := #I_AlarmResetPB, PT := T#1s);   // TOF
END_REGION

REGION Network 29: **** 8 - Outputs **** Auto mode
   // Auto mode
   #O_Auto := #Auto;
END_REGION

REGION Network 30: **** 8 - Outputs **** Manual mode
   // Manual mode
   #O_Man := #Man;
END_REGION

REGION Network 31: **** 8 - Outputs **** Auto selected mode
   // Auto selected mode
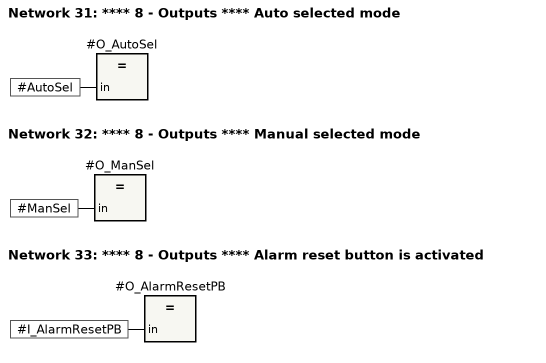
   #O_AutoSel := #AutoSel;
END_REGION

REGION Network 32: **** 8 - Outputs **** Manual selected mode
   // Manual selected mode
   #O_ManSel := #ManSel;
END_REGION

REGION Network 33: **** 8 - Outputs **** Alarm reset button is activated
   // Alarm reset button is activated
   #O_AlarmResetPB := #I_AlarmResetPB;
END_REGION
END_FUNCTION_BLOCK
